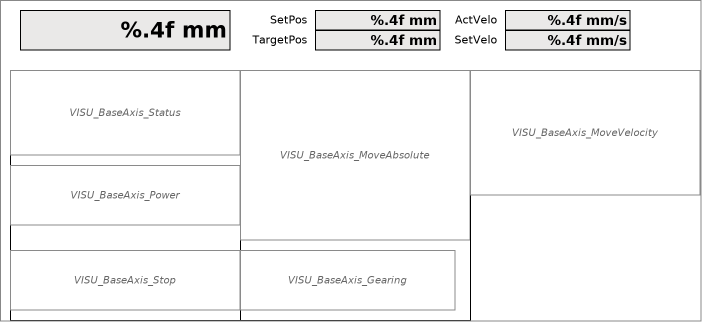
VISUALIZATION VISU_LinearAxis  // 702x322
VAR_IN_OUT
	axis : LinearAxis;
	widget : LinearAxisWidget;
END_VAR
    Rectangle (20,10 210x40), "%.4f mm", text variable: axis.actPos.millimeters.value
    Line (240,80) (240,320)
    Line (10,80) (10,320)
    Line (10,320) (470,320)
    Frame (10,70 230x85)
        shows VISU_BaseAxis_Status(axis := axis, axisWidget := widget.base)
    Frame (10,165 230x60)
        shows VISU_BaseAxis_Power(axis := axis, axisWidget := widget.base)
    Frame (240,70 230x170)
        shows VISU_BaseAxis_MoveAbsolute(axis := axis, axisWidget := widget.base, positionSymbol := widget.positionSymbol, velocitySymbol := widget.velocitySymbol)
    Frame (10,250 230x60)
        shows VISU_BaseAxis_Stop(axis := axis, axisWidget := widget.base)
    Line (470,80) (470,320)
    Frame (240,250 215x60)
        shows VISU_BaseAxis_Gearing(axis := axis, axisWidget := widget.base)
    Frame (470,70 230x125)
        shows VISU_BaseAxis_MoveVelocity(axis := axis, axisWidget := widget.base, positionSymbol := widget.positionSymbol, velocitySymbol := widget.velocitySymbol)
    Rectangle (315,10 125x20), "%.4f mm", text variable: axis.axis_ref.NcToPlc.SetPos
    Label (260,10 50x20), "SetPos"
    Rectangle (315,30 125x20), "%.4f mm", text variable: axis.axis_ref.NcToPlc.TargetPos
    Label (245,30 65x20), "TargetPos"
    Rectangle (505,10 125x20), "%.4f mm/s", text variable: axis.axis_ref.NcToPlc.ActVelo
    Label (450,10 50x20), "ActVelo"
    Label (450,30 50x20), "SetVelo"
    Rectangle (505,30 125x20), "%.4f mm/s", text variable: axis.axis_ref.NcToPlc.SetVelo
END_VISUALIZATION

(* stored: Version 1.1.0.1, ProductVersion 3.1.4019.2
   Visu VISU_LinearAxis: Id {31293ee7-a084-46c0-9ca7-1b893d37015c} *)
